Universal Robots PolyScope program: Arla0.7.urp

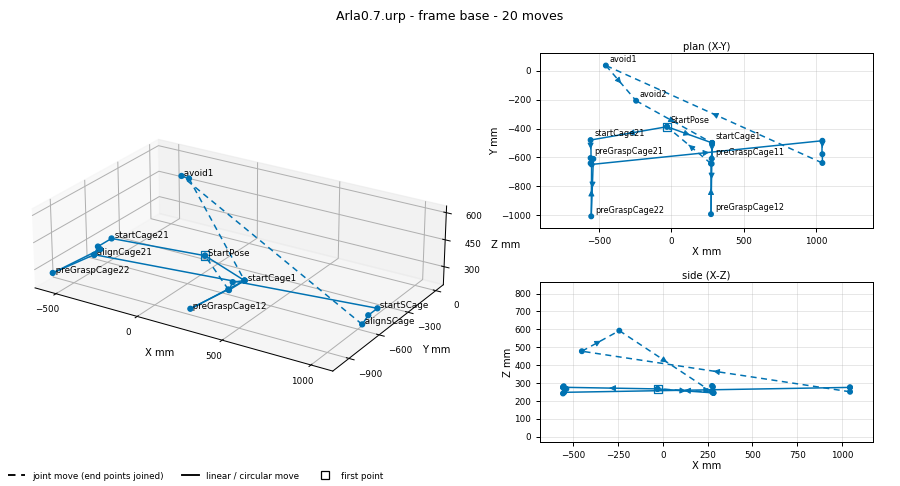
[picture p0: tool path of Arla0.7.urp in frame base, 20 of 20 moves have a stored position in this frame; points joined in program order, loops and branches not executed]
Program Arla0.7 (installation=default directory=/home/asger/Downloads/ursim-5.11.4.108353/programs/testArla createdIn=5.11.4.108353 lastSavedIn=5.11.4.108353 robotSerialNumber=20195299999)
Calibrated DH parameters: a=[0, -0.6127, -0.57155, 0, 0, 0]; d=[0.1807, 0, 0, 0.17415, 0.11985, 0.11655]; alpha=[1.570796, 0, 0, 1.570796, -1.570796, 0]; deltaTheta=[0, 0, 0, 0, 0, 0]
Robot Program (runOnlyOnce=true)
  Folder resetForce
    Wait Condition expression=is_steady()
    Wait Sleep waitTime=0.25
    Script: zero_ftsensor()
    Wait Sleep waitTime=0.25
  Timer (action=Start) variable(name=timer_1)
  MoveJ speed 30 deg/s, acceleration 40 deg/s^2 (useActiveTCP=true) feature=Base
    Waypoint StartPose: motionParameters(jointSpeed=0.523599 jointAcceleration=0.698132 cartesianSpeed=0.25 cartesianAcceleration=1.2); TCP in base x=-29.649 y=-387.378 z=267.725 mm, rx=0 ry=-3.1416 rz=0 rad; joints [-67.884, -70.586, -150.404, -49.041, 89.902, 22.237] deg
  Folder cage1
    MoveL speed 250 mm/s, acceleration 1200 mm/s^2 (useActiveTCP=true) feature=Base
      Waypoint startCage1: TCP in base x=282.101 y=-499.191 z=245.478 mm, rx=-0.1424 ry=-3.1383 rz=0 rad; joints [-42.958, -94.686, -134.076, -41.273, 89.848, 52.336] deg
    MoveL speed 250 mm/s, acceleration 1200 mm/s^2 (useActiveTCP=true) feature=Base
      Waypoint preGraspCage11: TCP in base x=279.409 y=-608.238 z=278.94 mm, rx=-0.1414 ry=-3.1151 rz=-0.3008 rad; joints [-51.575, -100.793, -119.743, -58.165, 96.643, 43.231] deg
    MoveL speed 100 mm/s, acceleration 1200 mm/s^2 (useActiveTCP=true) feature=Base
      MoveDirectionNode (selectedDirection=YMinus)
        Until TOOL_CONTACT_DETECTION (allowActions=false retraction=0.005 decelerationAcceleration=3 decelerationAngularAcceleration=34.906585)
    MoveL speed 250 mm/s, acceleration 1200 mm/s^2 (useActiveTCP=true) feature=Base
      MoveDirectionNode (selectedDirection=ZPlus)
        Until DISTANCE (allowActions=false deceleration=3 distanceNodeType=STOP) Distance=0.02; motionParameters(blendRadius=0)
    MoveL speed 250 mm/s, acceleration 1200 mm/s^2 (useActiveTCP=true) feature=Base
      Waypoint alignCage11: TCP in base x=279.344 y=-643.281 z=248.427 mm, rx=-0.1423 ry=-3.1374 rz=0 rad; joints [-52.242, -105.071, -120.426, -44.567, 89.777, 43.038] deg
    Set DigitalOutput pin=digital_out[0]; digitalValue=1
    Wait Sleep waitTime=0.7
    var_1 := get_actual_tcp_pose()
    Force Frame feature=Base; selection=[0, 0, 1, 0, 0, 0]; wrench=[0, 10, 225, 0, 0, 0]; limitsForce=[0.15, 0.15, 0.15, 1.047198, 1.047198, 1.047198]; limitsMotion=[0.1, 0.1, 0.1, 0.349066, 0.349066, 0.349066]
      Loop While (checkContinuously=false) expression=var_1[2] < 0.275
        var_1 := get_actual_tcp_pose()
    MoveL speed 100 mm/s, acceleration 1200 mm/s^2 (useActiveTCP=true) feature=Base
      MoveDirectionNode (selectedDirection=YPlus)
        Until DISTANCE (allowActions=false deceleration=3 distanceNodeType=STOP) Distance=0.1; motionParameters(blendRadius=0)
    Set DigitalOutput pin=digital_out[0]; digitalValue=0
    MoveL speed 100 mm/s, acceleration 1200 mm/s^2 (useActiveTCP=true) feature=Base
      MoveDirectionNode (selectedDirection=YPlus)
        Until DISTANCE (allowActions=false deceleration=3 distanceNodeType=BLEND) Distance=0.25; motionParameters(blendRadius=0)
    MoveL speed 200 mm/s, acceleration 400 mm/s^2 (useActiveTCP=true) feature=Base
      MoveDirectionNode (selectedDirection=ZMinus)
        Until DISTANCE (allowActions=false deceleration=3 distanceNodeType=STOP) Distance=0.012; motionParameters(blendRadius=0)
    MoveL speed 200 mm/s, acceleration 400 mm/s^2 (useActiveTCP=true) feature=Base
      MoveDirectionNode (selectedDirection=YPlus)
        Until DISTANCE (allowActions=false deceleration=3 distanceNodeType=STOP) Distance=0.085; motionParameters(blendRadius=0)
    MoveL speed 200 mm/s, acceleration 400 mm/s^2 (useActiveTCP=true) feature=Base
      MoveDirectionNode (selectedDirection=ZMinus)
        Until DISTANCE (allowActions=false deceleration=3 distanceNodeType=STOP) Distance=0.025; motionParameters(blendRadius=0)
    MoveL speed 200 mm/s, acceleration 400 mm/s^2 (useActiveTCP=true) feature=Base
      MoveDirectionNode (selectedDirection=YPlus)
        Until DISTANCE (allowActions=false deceleration=3 distanceNodeType=STOP) Distance=0.05; motionParameters(blendRadius=0)
    Halt
    MoveL speed 250 mm/s, acceleration 1200 mm/s^2 (useActiveTCP=true) feature=Base
      Waypoint startCage1: TCP in base x=282.101 y=-499.191 z=245.478 mm, rx=-0.1424 ry=-3.1383 rz=0 rad; joints [-42.958, -94.686, -134.076, -41.273, 89.848, 52.336] deg
    MoveL speed 250 mm/s, acceleration 1200 mm/s^2 (useActiveTCP=true) feature=Base
      Waypoint preGraspCage12: TCP in base x=274.587 y=-991.614 z=284.495 mm, rx=0.1352 ry=3.1015 rz=0.3905 rad; joints [-65.64, -130.563, -72.376, -79.598, 96.795, 28.715] deg
    MoveL speed 100 mm/s, acceleration 1200 mm/s^2 (useActiveTCP=true) feature=Base
      MoveDirectionNode (selectedDirection=YMinus)
        Until TOOL_CONTACT_DETECTION (allowActions=false retraction=0.005 decelerationAcceleration=3 decelerationAngularAcceleration=34.906585)
    MoveL speed 250 mm/s, acceleration 1200 mm/s^2 (useActiveTCP=true) feature=Base
      MoveDirectionNode (selectedDirection=ZPlus)
        Until DISTANCE (allowActions=false deceleration=3 distanceNodeType=STOP) Distance=0.02; motionParameters(blendRadius=0)
    MoveL speed 250 mm/s, acceleration 1200 mm/s^2 (useActiveTCP=true) feature=Base
      MoveDirectionNode (selectedDirection=XPlus)
        Until DISTANCE (allowActions=false deceleration=3 distanceNodeType=STOP) Distance=0.03; motionParameters(blendRadius=0)
    MoveL speed 250 mm/s, acceleration 1200 mm/s^2 (useActiveTCP=true) feature=Base
      MoveDirectionNode (selectedDirection=XMinus)
        Until DISTANCE (allowActions=false deceleration=3 distanceNodeType=STOP) Distance=0.06; motionParameters(blendRadius=0)
    MoveL speed 250 mm/s, acceleration 1200 mm/s^2 (useActiveTCP=true) feature=Base
      MoveDirectionNode (selectedDirection=XPlus)
        Until DISTANCE (allowActions=false deceleration=3 distanceNodeType=STOP) Distance=0.03; motionParameters(blendRadius=0)
    MoveL speed 250 mm/s, acceleration 1200 mm/s^2 (useActiveTCP=true) feature=Base
      Waypoint alignCage12: TCP in base x=274.592 y=-642.103 z=250.521 mm, rx=0.1324 ry=3.1167 rz=0 rad; joints [-52.671, -104.726, -120.866, -43.625, 90.791, 42.285] deg
    Set DigitalOutput pin=digital_out[0]; digitalValue=1
    Wait Sleep waitTime=0.7
    var_1 := get_actual_tcp_pose()
    Force Frame feature=Base; selection=[0, 0, 1, 0, 0, 0]; wrench=[0, 10, 225, 0, 0, 0]; limitsForce=[0.15, 0.15, 0.15, 1.047198, 1.047198, 1.047198]; limitsMotion=[0.1, 0.1, 0.1, 0.349066, 0.349066, 0.349066]
      Loop While (checkContinuously=false) expression=var_1[2] < 0.2685
        var_1 := get_actual_tcp_pose()
    MoveL speed 100 mm/s, acceleration 1200 mm/s^2 (useActiveTCP=true) feature=Base
      MoveDirectionNode (selectedDirection=YPlus)
        Until DISTANCE (allowActions=false deceleration=3 distanceNodeType=STOP) Distance=0.1; motionParameters(blendRadius=0)
    Set DigitalOutput pin=digital_out[0]; digitalValue=0
    MoveL speed 100 mm/s, acceleration 1200 mm/s^2 (useActiveTCP=true) feature=Base
      MoveDirectionNode (selectedDirection=YPlus)
        Until DISTANCE (allowActions=false deceleration=3 distanceNodeType=BLEND) Distance=0.25; motionParameters(blendRadius=0)
    MoveL speed 200 mm/s, acceleration 400 mm/s^2 (useActiveTCP=true) feature=Base
      MoveDirectionNode (selectedDirection=ZMinus)
        Until DISTANCE (allowActions=false deceleration=3 distanceNodeType=STOP) Distance=0.012; motionParameters(blendRadius=0)
    MoveL speed 200 mm/s, acceleration 400 mm/s^2 (useActiveTCP=true) feature=Base
      MoveDirectionNode (selectedDirection=YPlus)
        Until DISTANCE (allowActions=false deceleration=3 distanceNodeType=STOP) Distance=0.085; motionParameters(blendRadius=0)
    MoveL speed 200 mm/s, acceleration 400 mm/s^2 (useActiveTCP=true) feature=Base
      MoveDirectionNode (selectedDirection=ZMinus)
        Until DISTANCE (allowActions=false deceleration=3 distanceNodeType=STOP) Distance=0.02; motionParameters(blendRadius=0)
    MoveL speed 200 mm/s, acceleration 400 mm/s^2 (useActiveTCP=true) feature=Base
      MoveDirectionNode (selectedDirection=YPlus)
        Until DISTANCE (allowActions=false deceleration=3 distanceNodeType=STOP) Distance=0.05; motionParameters(blendRadius=0)
    Halt
    Wait Sleep waitTime=2
  MoveJ speed 30 deg/s, acceleration 40 deg/s^2 (useActiveTCP=true) feature=Base
    Waypoint StartPose: motionParameters(jointSpeed=0.523599 jointAcceleration=0.698132 cartesianSpeed=0.25 cartesianAcceleration=1.2); TCP in base x=-29.649 y=-387.378 z=267.725 mm, rx=0 ry=-3.1416 rz=0 rad; joints [-67.884, -70.586, -150.404, -49.041, 89.902, 22.237] deg
  Halt
  Folder cage2
    MoveL speed 250 mm/s, acceleration 1200 mm/s^2 (useActiveTCP=true) feature=Base
      Waypoint startCage21: TCP in base x=-557.376 y=-479.416 z=276.82 mm, rx=0.0973 ry=3.1401 rz=0 rad; joints [-125.598, -105.637, -115.68, -48.683, 90, -32.048] deg
    MoveL speed 250 mm/s, acceleration 1200 mm/s^2 (useActiveTCP=true) feature=Base
      Waypoint preGraspCage21: TCP in base x=-557.376 y=-603.558 z=276.82 mm, rx=0.0973 ry=3.1241 rz=0.3128 rad; joints [-119.809, -112.93, -102.706, -64.532, 84.453, -25.635] deg
    MoveL speed 100 mm/s, acceleration 1200 mm/s^2 (useActiveTCP=true) feature=Base
      MoveDirectionNode (selectedDirection=YMinus)
        Until TOOL_CONTACT_DETECTION (allowActions=false retraction=0.005 decelerationAcceleration=3 decelerationAngularAcceleration=34.906585)
    MoveL speed 250 mm/s, acceleration 1200 mm/s^2 (useActiveTCP=true) feature=Base
      MoveDirectionNode (selectedDirection=ZPlus)
        Until DISTANCE (allowActions=false deceleration=3 distanceNodeType=STOP) Distance=0.02; motionParameters(blendRadius=0)
    MoveL speed 250 mm/s, acceleration 1200 mm/s^2 (useActiveTCP=true) feature=Base
      Waypoint alignCage21: TCP in base x=-557.337 y=-639.505 z=242.248 mm, rx=0.0969 ry=3.134 rz=-0.0001 rad; joints [-119.351, -116.672, -103.581, -49.934, 90.088, -25.735] deg
    Set DigitalOutput pin=digital_out[0]; digitalValue=1
    Wait Sleep waitTime=0.7
    var_1 := get_actual_tcp_pose()
    Force Frame feature=Base; selection=[0, 0, 1, 0, 0, 0]; wrench=[0, 10, 225, 0, 0, 0]; limitsForce=[0.15, 0.15, 0.15, 1.047198, 1.047198, 1.047198]; limitsMotion=[0.1, 0.1, 0.1, 0.349066, 0.349066, 0.349066]
      Loop While (checkContinuously=false) expression=var_1[2] < 0.2685
        var_1 := get_actual_tcp_pose()
    MoveL speed 250 mm/s, acceleration 1200 mm/s^2 (useActiveTCP=true) feature=Base
      MoveDirectionNode (selectedDirection=YPlus)
        Until DISTANCE (allowActions=false deceleration=3 distanceNodeType=STOP) Distance=0.1; motionParameters(blendRadius=0)
    Set DigitalOutput pin=digital_out[0]; digitalValue=0
    MoveL speed 100 mm/s, acceleration 1200 mm/s^2 (useActiveTCP=true) feature=Base
      MoveDirectionNode (selectedDirection=YPlus)
        Until DISTANCE (allowActions=false deceleration=3 distanceNodeType=STOP) Distance=0.25; motionParameters(blendRadius=0)
    MoveL speed 200 mm/s, acceleration 400 mm/s^2 (useActiveTCP=true) feature=Base
      MoveDirectionNode (selectedDirection=ZMinus)
        Until DISTANCE (allowActions=false deceleration=3 distanceNodeType=STOP) Distance=0.012; motionParameters(blendRadius=0)
    MoveL speed 200 mm/s, acceleration 400 mm/s^2 (useActiveTCP=true) feature=Base
      MoveDirectionNode (selectedDirection=YPlus)
        Until DISTANCE (allowActions=false deceleration=3 distanceNodeType=STOP) Distance=0.085; motionParameters(blendRadius=0)
    MoveL speed 200 mm/s, acceleration 400 mm/s^2 (useActiveTCP=true) feature=Base
      MoveDirectionNode (selectedDirection=ZMinus)
        Until DISTANCE (allowActions=false deceleration=3 distanceNodeType=STOP) Distance=0.02; motionParameters(blendRadius=0)
    MoveL speed 200 mm/s, acceleration 400 mm/s^2 (useActiveTCP=true) feature=Base
      MoveDirectionNode (selectedDirection=YPlus)
        Until DISTANCE (allowActions=false deceleration=3 distanceNodeType=STOP) Distance=0.05; motionParameters(blendRadius=0)
    Halt
    MoveL speed 250 mm/s, acceleration 1200 mm/s^2 (useActiveTCP=true) feature=Base
      Waypoint startCage22: TCP in base x=-538.347 y=-609.44 z=268.172 mm, rx=0.0966 ry=3.1337 rz=0.0061 rad; joints [-119.209, -112.389, -106.906, -51.102, 90.007, -25.595] deg
    MoveL speed 400 mm/s, acceleration 1200 mm/s^2 (useActiveTCP=true) feature=Base
      Waypoint preGraspCage22: TCP in base x=-552.966 y=-1006.741 z=282.788 mm, rx=0.0951 ry=3.1094 rz=0.4082 rad; joints [-109.644, -142.955, -49.635, -91.779, 85.364, -15.442] deg
    MoveL speed 100 mm/s, acceleration 1200 mm/s^2 (useActiveTCP=true) feature=Base
      MoveDirectionNode (selectedDirection=YMinus)
        Until TOOL_CONTACT_DETECTION (allowActions=false retraction=0.005 decelerationAcceleration=3 decelerationAngularAcceleration=34.906585)
    MoveL speed 250 mm/s, acceleration 1200 mm/s^2 (useActiveTCP=true) feature=Base
      MoveDirectionNode (selectedDirection=ZPlus)
        Until DISTANCE (allowActions=false deceleration=3 distanceNodeType=STOP) Distance=0.02; motionParameters(blendRadius=0)
    MoveL speed 250 mm/s, acceleration 1200 mm/s^2 (useActiveTCP=true) feature=Base
      MoveDirectionNode (selectedDirection=XPlus)
        Until DISTANCE (allowActions=false deceleration=3 distanceNodeType=STOP) Distance=0.025; motionParameters(blendRadius=0)
    MoveL speed 250 mm/s, acceleration 1200 mm/s^2 (useActiveTCP=true) feature=Base
      MoveDirectionNode (selectedDirection=XMinus)
        Until DISTANCE (allowActions=false deceleration=3 distanceNodeType=STOP) Distance=0.05; motionParameters(blendRadius=0)
    MoveL speed 250 mm/s, acceleration 1200 mm/s^2 (useActiveTCP=true) feature=Base
      MoveDirectionNode (selectedDirection=XPlus)
        Until DISTANCE (allowActions=false deceleration=3 distanceNodeType=STOP) Distance=0.025; motionParameters(blendRadius=0)
    MoveL speed 400 mm/s, acceleration 1200 mm/s^2 (useActiveTCP=true) feature=Base
      Waypoint alignCage22: TCP in base x=-550.35 y=-647.871 z=248.708 mm, rx=0.0972 ry=3.1358 rz=-0.0001 rad; joints [-118.638, -116.404, -103.185, -50.55, 89.996, -25.012] deg
    var_1 := get_actual_tcp_pose()
    Force Frame feature=Base; selection=[0, 0, 1, 0, 0, 0]; wrench=[0, 10, 225, 0, 0, 0]; limitsForce=[0.15, 0.15, 0.15, 1.047198, 1.047198, 1.047198]; limitsMotion=[0.1, 0.1, 0.1, 0.349066, 0.349066, 0.349066]
      Loop While (checkContinuously=false) expression=var_1[2] < 0.2685
        var_1 := get_actual_tcp_pose()
    Wait Sleep waitTime=0.7
    MoveL speed 200 mm/s, acceleration 400 mm/s^2 (useActiveTCP=true) feature=Base
      MoveDirectionNode (selectedDirection=YPlus)
        Until DISTANCE (allowActions=false deceleration=3 distanceNodeType=STOP) Distance=0.25; motionParameters(blendRadius=0.05)
    MoveL speed 100 mm/s, acceleration 400 mm/s^2 (useActiveTCP=true) feature=Base
      MoveDirectionNode (selectedDirection=ZMinus)
        Until DISTANCE (allowActions=false deceleration=3 distanceNodeType=STOP) Distance=0.015; motionParameters(blendRadius=0)
    MoveL speed 200 mm/s, acceleration 400 mm/s^2 (useActiveTCP=true) feature=Base
      MoveDirectionNode (selectedDirection=YPlus)
        Until DISTANCE (allowActions=false deceleration=3 distanceNodeType=STOP) Distance=0.185; motionParameters(blendRadius=0)
    MoveL speed 200 mm/s, acceleration 400 mm/s^2 (useActiveTCP=true) feature=Base
      MoveDirectionNode (selectedDirection=ZMinus)
        Until DISTANCE (allowActions=false deceleration=3 distanceNodeType=STOP) Distance=0.02; motionParameters(blendRadius=0)
    MoveL speed 200 mm/s, acceleration 400 mm/s^2 (useActiveTCP=true) feature=Base
      MoveDirectionNode (selectedDirection=YPlus)
        Until DISTANCE (allowActions=false deceleration=3 distanceNodeType=STOP) Distance=0.05; motionParameters(blendRadius=0)
    Halt
  Timer (action=Stop) variable=timer_1
  Folder sCage
    MoveL speed 250 mm/s, acceleration 1200 mm/s^2 (useActiveTCP=true) feature=Base
      Waypoint startSCage: TCP in base x=1044.119 y=-484.269 z=276.229 mm, rx=0.1134 ry=3.1395 rz=0 rad; joints [-16.179, -140.694, -57.245, -72.061, 90, 77.956] deg
    MoveL speed 250 mm/s, acceleration 1200 mm/s^2 (useActiveTCP=true) feature=Base
      Waypoint preGraspSCage: TCP in base x=1044.119 y=-577.153 z=276.229 mm, rx=-0.1134 ry=-3.1179 rz=-0.3018 rad; joints [-21.554, -146.793, -45.014, -82.317, 99.954, 72.324] deg
    MoveL speed 100 mm/s, acceleration 1200 mm/s^2 (useActiveTCP=true) feature=Base
      MoveDirectionNode (selectedDirection=YMinus)
        Until TOOL_CONTACT_DETECTION (allowActions=false retraction=0.005 decelerationAcceleration=3 decelerationAngularAcceleration=34.906585)
    MoveL speed 250 mm/s, acceleration 1200 mm/s^2 (useActiveTCP=true) feature=Base
      Waypoint alignSCage: TCP in base x=1044.334 y=-637.926 z=251.735 mm, rx=0.1158 ry=3.1385 rz=0 rad; joints [-23.245, -150.282, -41.443, -78.254, 89.697, 71.035] deg
    Set DigitalOutput pin=digital_out[0]; digitalValue=1
    Wait Sleep waitTime=0.7
    var_1 := get_actual_tcp_pose()
    Force Frame feature=Base; selection=[0, 0, 1, 0, 0, 0]; wrench=[0, 10, 225, 0, 0, 0]; limitsForce=[0.15, 0.15, 0.15, 1.047198, 1.047198, 1.047198]; limitsMotion=[0.1, 0.1, 0.1, 0.349066, 0.349066, 0.349066]
      Loop While (checkContinuously=false) expression=var_1[2] < 0.2685
        var_1 := get_actual_tcp_pose()
    MoveL speed 250 mm/s, acceleration 1200 mm/s^2 (useActiveTCP=true) feature=Base
      MoveDirectionNode (selectedDirection=YPlus)
        Until DISTANCE (allowActions=false deceleration=3 distanceNodeType=STOP) Distance=0.1; motionParameters(blendRadius=0)
    Set DigitalOutput pin=digital_out[0]; digitalValue=0
    MoveL speed 100 mm/s, acceleration 1200 mm/s^2 (useActiveTCP=true) feature=Base
      MoveDirectionNode (selectedDirection=YPlus)
        Until DISTANCE (allowActions=false deceleration=3 distanceNodeType=STOP) Distance=0.25; motionParameters(blendRadius=0)
    MoveL speed 200 mm/s, acceleration 400 mm/s^2 (useActiveTCP=true) feature=Base
      MoveDirectionNode (selectedDirection=ZMinus)
        Until DISTANCE (allowActions=false deceleration=3 distanceNodeType=STOP) Distance=0.012; motionParameters(blendRadius=0)
    MoveL speed 200 mm/s, acceleration 400 mm/s^2 (useActiveTCP=true) feature=Base
      MoveDirectionNode (selectedDirection=YPlus)
        Until DISTANCE (allowActions=false deceleration=3 distanceNodeType=STOP) Distance=0.085; motionParameters(blendRadius=0)
    MoveL speed 200 mm/s, acceleration 400 mm/s^2 (useActiveTCP=true) feature=Base
      MoveDirectionNode (selectedDirection=ZMinus)
        Until DISTANCE (allowActions=false deceleration=3 distanceNodeType=STOP) Distance=0.02; motionParameters(blendRadius=0)
    MoveL speed 200 mm/s, acceleration 400 mm/s^2 (useActiveTCP=true) feature=Base
      MoveDirectionNode (selectedDirection=YPlus)
        Until DISTANCE (allowActions=false deceleration=3 distanceNodeType=STOP) Distance=0.05; motionParameters(blendRadius=0)
  Folder avoidStack
    MoveJ speed 60 deg/s, acceleration 80 deg/s^2 (useActiveTCP=true) feature=Base
      Waypoint avoid1: TCP in base x=-451.899 y=35.465 z=478.022 mm, rx=0.229 ry=-2.3873 rz=-1.3939 rad; joints [-147.022, -61.498, -134.665, -88.432, 27.226, -58.848] deg
      Waypoint avoid2: TCP in base x=-242.971 y=-207.894 z=592.766 mm, rx=1.6853 ry=-1.4447 rz=-1.1258 rad; joints [-80.323, -39.086, -127.817, -129.874, 28.453, -72.722] deg
      Waypoint avoid3: TCP in base x=282.11 y=-499.2 z=245.477 mm, rx=-0.1425 ry=-3.1383 rz=-0.0001 rad; joints [-42.958, -94.687, -134.074, -41.273, 89.851, 52.338] deg
